PROGRAM PRG_Database
VAR
	fbSystemTime			: FB_SystemTime;
	bSaveData				: BOOL;
	bLoadData				: BOOL;
	nStateSave, nStateLoad	: INT;
	tTimer1, tTimer2		: TON;
	bTest					: BOOL;
	nStateADS				: INT;
END_VAR

fbSystemTime();
sCurrentTime	:= fbSystemTime.sTime;
nCurrentSec		:= fbSystemTime.wSecond;
CASE nStateSave OF
	0:
		tTimer1(IN := FALSE);
		IF nCurrentSec = 70 OR sCurrentTime = '06:00:00' OR sCurrentTime = '14:00:00' OR sCurrentTime = '22:00:00' THEN
			nStateSave			:= 1;
		END_IF
	1:
		aFFTU1						:= aSpectrum[0];
		aFFTU2						:= aSpectrum[1];
		aFFTU3						:= aSpectrum[2];
		
		aFFTI1						:= aSpectrum[3];
		aFFTI2						:= aSpectrum[4];
		aFFTI3						:= aSpectrum[5];
		
		RMSI1						:= MAIN.fbBasicValues.aRMS_I[0]/2.44;
		RMSI2						:= MAIN.fbBasicValues.aRMS_I[1]/2.44;
		RMSI3						:= MAIN.fbBasicValues.aRMS_I[2]/2.44;
		
		RMSU1						:= MAIN.fbBasicValues.aRMS_U[0];
		RMSU2						:= MAIN.fbBasicValues.aRMS_U[1];
		RMSU3						:= MAIN.fbBasicValues.aRMS_U[2];		
		
		Frequency					:= LREAL_TO_REAL(MAIN.fbFrequency.aFreq[0]);
		
		bAddData					:= TRUE;
		nStateSave					:= 2;
	2:
		IF NOT bAddData THEN
			tTimer1(IN := TRUE,PT := T#2S);
			IF tTimer1.Q THEN
				nStateSave			:= 0;		
			END_IF	
		END_IF
			
		
END_CASE

CASE nStateADS OF
	0:
		IF bCheckADS THEN
			nStateADS := 1;
		ELSE
			tTimer2(IN := TRUE,PT := T#5S);
			IF tTimer2.Q THEN
				nStateADS := 2;
			END_IF
		END_IF
		
	1:
		bCheckADS := FALSE;
		bError	:= FALSE;
		tTimer2(IN := FALSE);
		nStateADS := 0;
	2:
		bError := TRUE;
		tTimer2(IN := FALSE);
		IF bCheckADS THEN
			nStateADS := 0;
		END_IF
END_CASE

END_PROGRAM

(* stored: Version 1.1.0.1, ProductVersion 3.1.4024.12
   POU PRG_Database: Id {15ffa7de-2a8f-4618-b011-b02082bc35fe}, SpecialFunc None *)
